(* PLC project SafeLOGIC-1, BrAutomation SafeDESIGNER  4.3.2.11 *)
(* stored: companyURL http://www.br-automation.com, creationDateTime Tue Mar 06 09:58:23 2018 *)

PROGRAM Main

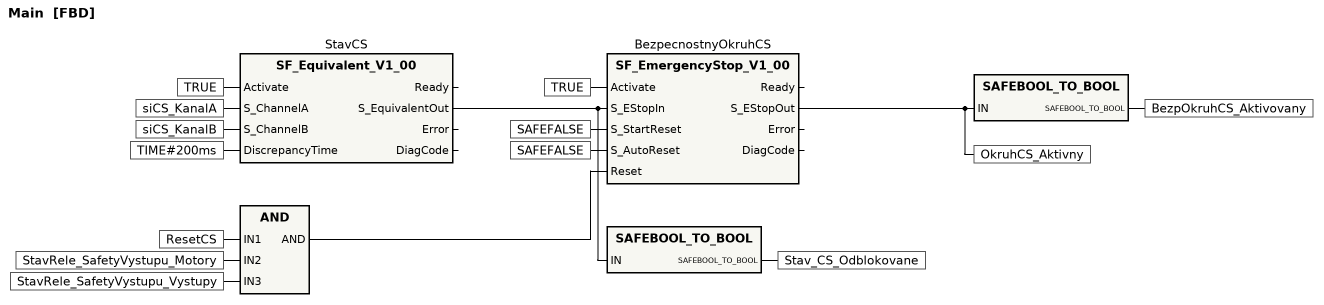
(* FBD diagram, written out as Structured Text *)
StavCS(Activate := TRUE, S_ChannelA := siCS_KanalA, S_ChannelB := siCS_KanalB, DiscrepancyTime := TIME#200ms);
BezpecnostnyOkruhCS(Activate := TRUE, S_EStopIn := StavCS.S_EquivalentOut, S_StartReset := SAFEFALSE, S_AutoReset := SAFEFALSE, Reset := ResetCS AND StavRele_SafetyVystupu_Motory AND StavRele_SafetyVystupu_Vystupy);
OkruhCS_Aktivny := BezpecnostnyOkruhCS.S_EStopOut;
Stav_CS_Odblokovane := SAFEBOOL_TO_BOOL(StavCS.S_EquivalentOut);
BezpOkruhCS_Aktivovany := SAFEBOOL_TO_BOOL(BezpecnostnyOkruhCS.S_EStopOut);
END_PROGRAM
